PROGRAM P_Demo_Execute
VAR
    fbListener : FB_ListenerBase2; // listener 实例
    hr         : HRESULT; // 返回值监视
END_VAR

// =============================================================================
// 场景：主程序里每周期推进事件队列
// 价值：必须周期调用以保证事件及时到达回调
// 验证：登录后 monitor hr，每周期应为 S_OK；fbListener 必须已 Subscribe
// 验证步骤：
//   1. 右键 PLC 项目下 POUs 文件夹 → Add → Existing Item → 选本 .TcPOU 文件
//   2. 引用 Tc3_EventLogger（System → References → Add library）
//   3. 编译 → 登录 → 运行；按 verify 注释里给出的在线写值操作
// =============================================================================

// 每周期调用一次推进事件队列
hr := fbListener.Execute();

END_PROGRAM

(* stored: Version 1.1.0.1, ProductVersion 3.1.4024.5
   POU P_Demo_Execute: Id {e67d2fad-61b3-5158-bbcb-d5df361ad5fc}, SpecialFunc None *)
